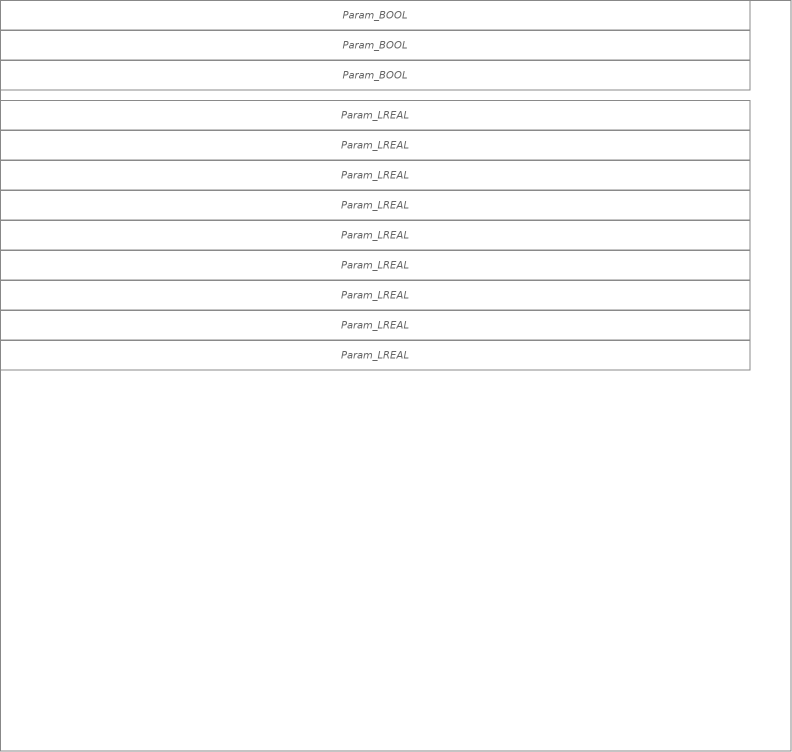
VISUALIZATION Visu_Mparam_Autotune  // 792x752
    Frame (0,100 750x30)
        shows Param_LREAL(nIdx := 24)
    Frame (0,130 750x30)
        shows Param_LREAL(nIdx := 25)
    Frame (0,160 750x30)
        shows Param_LREAL(nIdx := 26)
    Frame (0,190 750x30)
        shows Param_LREAL(nIdx := 27)
    Frame (0,220 750x30)
        shows Param_LREAL(nIdx := 28)
    Frame (0,250 750x30)
        shows Param_LREAL(nIdx := 29)
    Frame (0,280 750x30)
        shows Param_LREAL(nIdx := 30)
    Frame (0,310 750x30)
        shows Param_LREAL(nIdx := 31)
    Frame (0,340 750x30)
        shows Param_LREAL(nIdx := 23)
    Frame (0,60 750x30)
        shows Param_BOOL(nIdx := 10)
    Frame (0,30 750x30)
        shows Param_BOOL(nIdx := 4)
    Frame (0,0 750x30)
        shows Param_BOOL(nIdx := 5)
    Rectangle (40,720 750x30)
END_VISUALIZATION

(* stored: Version 1.1.0.1
   Visu Visu_Mparam_Autotune: Id {0a55b6fb-9821-48ff-960b-1eabb1dd498e} *)
